// TIA Portal V16 export
// export: Created 2022-11-17T11:55:30.5376514Z, ExportSetting WithDefaults, DisplayName Totally Integrated Automation Portal, DisplayVersion V16 Update 6, DisplayName TIA Portal Version Control Interface, DisplayVersion V16 Update 2, DisplayName TIA Portal Openness, DisplayVersion V16 Update 6, DisplayName SINAMICS Startdrive Advanced, DisplayVersion V16 Update 5, DisplayName SINAMICS Startdrive G130, G150, S120, S150, SINAMICS MV, S210, DisplayVersion V16 Update 5, DisplayName SINAMICS Startdrive G110M, G120, G120C, G120D, G120P, G115D, DisplayVersion V16 Update 5, DisplayName STEP 7 Professional, DisplayVersion V16 Update 6, DisplayName STEP 7 Safety, DisplayVersion V16, DisplayName WinCC Advanced, DisplayVersion V16 Update 6
DATA_BLOCK "DB100_Display"   // DB100
{ S7_Optimized_Access := 'FALSE' }
VERSION : 0.1
// stored: AutoNumber false, IsOnlyStoredInLoadMemory false, IsWriteProtectedInAS false
   VAR RETAIN
      CELLA : Int := 15;   // CELLA (rosa)
      SETPOINT : UInt := 20;   // SETPOINT (rosso)
      PROP : Int := 0;   // PROPORZIONALE (verde)
      "INT" : Int := 0;   // INTEGRALE (giallo)
      FREQ_TIRO : Int := 0;   // U241
      FREQ_PRES : Int := 0;   // U261
   END_VAR
BEGIN
END_DATA_BLOCK
